// TIA Portal V17 export
// export: Created 2025-03-07T09:24:32.6237895Z, ExportSetting WithDefaults, DisplayName Totally Integrated Automation Portal, DisplayVersion V17 Update 8, DisplayName TIA Portal Openness, DisplayVersion V17 Update 8, DisplayName TIA Portal Version Control Interface, DisplayVersion V17, DisplayName SINAMICS Startdrive Advanced, DisplayVersion V17 SP2, DisplayName SINAMICS Startdrive G110M, G120, G120C, G120D, G120P, G115D, DisplayVersion V17 SP2, DisplayName SINAMICS Startdrive G130, G150, S120, S150, SINAMICS MV, S210, DisplayVersion V17 SP2, DisplayName STEP 7 Professional, DisplayVersion V17 Update 8, DisplayName SINUMERIK ONE STEP 7 Toolbox, DisplayVersion V17 Update 12, DisplayName SINUMERIK 840D sl STEP 7 Toolbox, DisplayVersion V17 Update 12, DisplayName STEP 7 Safety, DisplayVersion V17 Update 6, DisplayName WinCC Advanced, DisplayVersion V17 Update 8
VAR_GLOBAL   // PLC tag table "TAGS_IO_STIRRERS_CLADDING"
   "//////////_STIRRER_UNIT_01_HOPPER_1_//////////" AT %M500.0 : Bool;
   "//////////_STIRRER_UNIT_01_HOPPER_2_//////////" AT %M600.0 : Bool;
   "//////////_STIRRER_UNIT_02_HOPPER_1_//////////" AT %M2000.0 : Bool;
   "//////////_STIRRER_UNIT_02_HOPPER_2_//////////" AT %M800.0 : Bool;
   "//////////_STIRRER_UNIT_02_HOPPER_3_//////////" AT %M900.0 : Bool;
   U01_HPPR_1_STRR_ACTUAL_PHASE_CURRENT_FILTERED_INPUT AT %ID3016 : DInt;   // UNIT 01 HOPPER 1 STIRRER ACTUAL PHASE CURRENT FILTERED INPUT
   U01_HPPR_1_STRR_ACTUAL_PHASE_CURRENT_INPUT AT %ID3012 : DInt;   // UNIT 01 HOPPER 1 STIRRER ACTUAL PHASE CURRENT INPUT
   U01_HPPR_1_STRR_ACTUAL_POSITION_INPUT AT %ID3008 : DInt;   // UNIT 01 HOPPER 1 STIRRER STIRRER ACTUAL POSITON INPUT
   U01_HPPR_1_STRR_ACTUAL_TEMP_COM AT %IW3023 : Int;   // UNIT 01 HOPPER 1 STIRRER ACTUAL COM CARD TEMPERATURE
   U01_HPPR_1_STRR_ACTUAL_TEMP_POWER AT %IW3021 : Int;   // UNIT 01 HOPPER 1 STIRRER ACTUAL POWER STAGE TEMPERATURE
   U01_HPPR_1_STRR_ACTUAL_VELOCITY_INPUT AT %ID3004 : DInt;   // UNIT 01 HOPPER 1 STIRRER ACTUAL VELOCITY INPUT
   U01_HPPR_1_STRR_ENABLE_POWER_STAGE_OUTPUT AT %QB3005 : Byte;   // UNIT 01 HOPPER 1 STIRRER ENABLE POWER STAGE
   U01_HPPR_1_STRR_ERROR_CODE AT %IW3025 : Int;   // UNIT 01 HOPPER 1 STIRRER ERROR CODE
   U01_HPPR_1_STRR_IO_DIGITAL_OUTPUTS AT %QB3000 : Byte;   // UNIT 01 HOPPER 1 STIRRER IO DIGITAL OUTPUTS
   U01_HPPR_1_STRR_MODE_OF_OPERATION_OUTPUT AT %QB3006 : Byte;   // UNIT 01 HOPPER 1 STIRRER MODE OF OPERATION OUTPUT
   U01_HPPR_1_STRR_MOTOR_ENABLE_1_Q AT %M500.1 : Bool;   // UNIT 01 HOPPER 1 STIRRER MOTOR ENABLE 1 OUTPUT
   U01_HPPR_1_STRR_MOTOR_ENABLE_2_Q AT %M500.2 : Bool;   // UNIT 01 HOPPER 1 STIRRER MOTOR ENABLE 2 OUTPUT
   U01_HPPR_1_STRR_MOTOR_OUT_1 AT %Q3000.1 : Bool;   // UNIT 01 HOPPER 1 STIRRER MOTOR OUT 1
   U01_HPPR_1_STRR_MOTOR_OUT_2 AT %Q3000.2 : Bool;   // UNIT 01 HOPPER 1 STIRRER MOTOR OUT 2
   U01_HPPR_1_STRR_MOTOR_OUT_3 AT %Q3000.3 : Bool;   // UNIT 01 HOPPER 1 STIRRER MOTOR OUT 3
   U01_HPPR_1_STRR_MOTOR_STATUS_ENABLE AT %I3020.0 : Bool;   // UNIT 01 HOPPER 1 STIRRER MOTOR STATUS ENABLED
   U01_HPPR_1_STRR_MOTOR_STATUS_ENABLE_INPUT AT %I3000.0 : Bool;   // UNIT 01 HOPPER 1 STIRRER MOTOR STATUS ENABLE INPUT
   U01_HPPR_1_STRR_MOTOR_STATUS_ERROR AT %I3020.1 : Bool;   // UNIT 01 HOPPER 1 STIRRER MOTOR STATUS ERROR
   U01_HPPR_1_STRR_MOTOR_STATUS_ERROR_INPUT AT %I3000.1 : Bool;   // UNIT 01 HOPPER 1 STIRRER MOTOR STATUS ERROR INPUT
   U01_HPPR_1_STRR_MOTOR_STATUS_REACHED AT %I3020.4 : Bool;   // UNIT 01 HOPPER 1 STIRRER MOTOR STATUS REACHED
   U01_HPPR_1_STRR_MOTOR_STATUS_REACHED_INPUT AT %I3000.4 : Bool;   // UNIT 01 HOPPER 1 STIRRER MOTOR STATUS REACHED INPUT
   U01_HPPR_1_STRR_POWER_STAGE_HW_ENABLE_INPUTS AT %IB3020 : Byte;   // UNIT 01 HOPPER 1 STIRRER POWER STAGE STAGE HW ENABLE INPUTS
   U01_HPPR_1_STRR_STATUS_REGISTER_INPUTS AT %ID3000 : DInt;   // UNIT 01 HOPPER 1 STIRRER STATUS REGISTER INPUTS
   U01_HPPR_2_STRR_ACTUAL_PHASE_CURRENT_FILTERED_INPUT AT %ID3116 : DInt;   // UNIT 01 HOPPER 2 STIRRER ACTUAL PHASE CURRENT FILTERED INPUT
   U01_HPPR_2_STRR_ACTUAL_PHASE_CURRENT_INPUT AT %ID3112 : DInt;   // UNIT 01 HOPPER 2 STIRRER ACTUAL PHASE CURRENT INPUT
   U01_HPPR_2_STRR_ACTUAL_POSITION_INPUT AT %ID3108 : DInt;   // UNIT 01 HOPPER 2 STIRRER STIRRER ACTUAL POSITON INPUT
   U01_HPPR_2_STRR_ACTUAL_TEMP_COM AT %IW3123 : Int;   // UNIT 01 HOPPER 2 STIRRER ACTUAL COM CARD TEMPERATURE
   U01_HPPR_2_STRR_ACTUAL_TEMP_POWER AT %IW3121 : Int;   // UNIT 01 HOPPER 2 STIRRER ACTUAL POWER STAGE TEMPERATURE
   U01_HPPR_2_STRR_ACTUAL_VELOCITY_INPUT AT %ID3104 : DInt;   // UNIT 01 HOPPER 2 STIRRER ACTUAL VELOCITY INPUT
   U01_HPPR_2_STRR_ENABLE_POWER_STAGE_OUTPUT AT %QB3105 : Byte;   // UNIT 01 HOPPER 2 STIRRER ENABLE POWER STAGE
   U01_HPPR_2_STRR_ERROR_CODE AT %IW3125 : Int;   // UNIT 01 HOPPER 2 STIRRER ERROR CODE
   U01_HPPR_2_STRR_IO_DIGITAL_OUTPUTS AT %QB3100 : Byte;   // UNIT 01 HOPPER 2 STIRRER IO DIGITAL OUTPUTS
   U01_HPPR_2_STRR_MODE_OF_OPERATION_OUTPUT AT %QB3106 : Byte;   // UNIT 01 HOPPER 2 STIRRER MODE OF OPERATION OUTPUT
   U01_HPPR_2_STRR_MOTOR_ENABLE_1_Q AT %M600.1 : Bool;   // UNIT 01 HOPPER 2 STIRRER MOTOR ENABLE 1 OUTPUT
   U01_HPPR_2_STRR_MOTOR_ENABLE_2_Q AT %M600.2 : Bool;   // UNIT 01 HOPPER 2 STIRRER MOTOR ENABLE 2 OUTPUT
   U01_HPPR_2_STRR_MOTOR_OUT_1 AT %Q3100.1 : Bool;   // UNIT 01 HOPPER 2 STIRRER MOTOR OUT 1
   U01_HPPR_2_STRR_MOTOR_OUT_2 AT %Q3100.2 : Bool;   // UNIT 01 HOPPER 2 STIRRER MOTOR OUT 2
   U01_HPPR_2_STRR_MOTOR_OUT_3 AT %Q3100.3 : Bool;   // UNIT 01 HOPPER 2 STIRRER MOTOR OUT 3
   U01_HPPR_2_STRR_MOTOR_STATUS_ENABLE AT %I3120.0 : Bool;   // UNIT 01 HOPPER 2 STIRRER MOTOR STATUS ENABLED
   U01_HPPR_2_STRR_MOTOR_STATUS_ENABLE_INPUT AT %I3100.0 : Bool;   // UNIT 01 HOPPER 2 STIRRER MOTOR STATUS ENABLE INPUT
   U01_HPPR_2_STRR_MOTOR_STATUS_ERROR AT %I3120.1 : Bool;   // UNIT 01 HOPPER 2 STIRRER MOTOR STATUS ERROR
   U01_HPPR_2_STRR_MOTOR_STATUS_ERROR_INPUT AT %I3100.1 : Bool;   // UNIT 01 HOPPER 2 STIRRER MOTOR STATUS ERROR INPUT
   U01_HPPR_2_STRR_MOTOR_STATUS_REACHED AT %I3120.4 : Bool;   // UNIT 01 HOPPER 2 STIRRER MOTOR STATUS REACHED
   U01_HPPR_2_STRR_MOTOR_STATUS_REACHED_INPUT AT %I3100.4 : Bool;   // UNIT 01 HOPPER 2 STIRRER MOTOR STATUS REACHED INPUT
   U01_HPPR_2_STRR_POWER_STAGE_HW_ENABLE_INPUTS AT %IB3120 : Byte;   // UNIT 01 HOPPER 2 STIRRER POWER STAGE STAGE HW ENABLE INPUTS
   U01_HPPR_2_STRR_STATUS_REGISTER_INPUTS AT %ID3100 : DInt;   // UNIT 01 HOPPER 2 STIRRER STATUS REGISTER INPUTS
   U01_HPPR_2_STRR_VEL_TARGET_VALUE_OUTPUT AT %QD3101 : DInt;   // UNIT 01 HOPPER 2 STIRRER VELOCITY TARGET VALUE OUTPUT
   U01_HPPR1_STRR_VEL_TARGET_VALUE_OUTPUT AT %QD3001 : DInt;   // UNIT 01 HOPPER 1 STIRRER VELOCITY TARGET VALUE OUTPUT
   U02_HPPR_1_STRR_ACTUAL_PHASE_CURRENT_FILTERED_INPUT AT %ID3216 : DInt;   // UNIT 02 HOPPER 1 STIRRER ACTUAL PHASE CURRENT FILTERED INPUT
   U02_HPPR_1_STRR_ACTUAL_PHASE_CURRENT_INPUT AT %ID3212 : DInt;   // UNIT 02 HOPPER 1 STIRRER ACTUAL PHASE CURRENT INPUT
   U02_HPPR_1_STRR_ACTUAL_POSITION_INPUT AT %ID3208 : DInt;   // UNIT 02 HOPPER 1 STIRRER STIRRER ACTUAL POSITON INPUT
   U02_HPPR_1_STRR_ACTUAL_TEMP_COM AT %IW3223 : Int;   // UNIT 02 HOPPER 1 STIRRER ACTUAL COM CARD TEMPERATURE
   U02_HPPR_1_STRR_ACTUAL_TEMP_POWER AT %IW3221 : Int;   // UNIT 02 HOPPER 1 STIRRER ACTUAL POWER STAGE TEMPERATURE
   U02_HPPR_1_STRR_ACTUAL_VELOCITY_INPUT AT %ID3204 : DInt;   // UNIT 02 HOPPER 1 STIRRER ACTUAL VELOCITY INPUT
   U02_HPPR_1_STRR_ENABLE_POWER_STAGE_OUTPUT AT %QB3205 : Byte;   // UNIT 02 HOPPER 1 STIRRER ENABLE POWER STAGE
   U02_HPPR_1_STRR_ERROR_CODE AT %IW3225 : Int;   // UNIT 02 HOPPER 1 STIRRER ERROR CODE
   U02_HPPR_1_STRR_IO_DIGITAL_OUTPUTS AT %QB3200 : Byte;   // UNIT 02 HOPPER 1 STIRRER IO DIGITAL OUTPUTS
   U02_HPPR_1_STRR_MODE_OF_OPERATION_OUTPUT AT %QB3206 : Byte;   // UNIT 02 HOPPER 1 STIRRER MODE OF OPERATION OUTPUT
   U02_HPPR_1_STRR_MOTOR_ENABLE_1_Q AT %M700.1 : Bool;   // UNIT 02 HOPPER 1 STIRRER MOTOR ENABLE 1 OUTPUT
   U02_HPPR_1_STRR_MOTOR_ENABLE_2_Q AT %M700.2 : Bool;   // UNIT 02 HOPPER 1 STIRRER MOTOR ENABLE 2 OUTPUT
   U02_HPPR_1_STRR_MOTOR_OUT_1 AT %Q3200.1 : Bool;   // UNIT 02 HOPPER 1 STIRRER MOTOR OUT 1
   U02_HPPR_1_STRR_MOTOR_OUT_2 AT %Q3200.2 : Bool;   // UNIT 02 HOPPER 1 STIRRER MOTOR OUT 2
   U02_HPPR_1_STRR_MOTOR_OUT_3 AT %Q3200.3 : Bool;   // UNIT 02 HOPPER 1 STIRRER MOTOR OUT 3
   U02_HPPR_1_STRR_MOTOR_STATUS_ENABLE AT %I3220.0 : Bool;   // UNIT 02 HOPPER 1 STIRRER MOTOR STATUS ENABLED
   U02_HPPR_1_STRR_MOTOR_STATUS_ENABLE_INPUT AT %I3200.0 : Bool;   // UNIT 02 HOPPER 1 STIRRER MOTOR STATUS ENABLE INPUT
   U02_HPPR_1_STRR_MOTOR_STATUS_ERROR AT %I3220.1 : Bool;   // UNIT 02 HOPPER 1 STIRRER MOTOR STATUS ERROR
   U02_HPPR_1_STRR_MOTOR_STATUS_ERROR_INPUT AT %I3200.1 : Bool;   // UNIT 02 HOPPER 1 STIRRER MOTOR STATUS ERROR INPUT
   U02_HPPR_1_STRR_MOTOR_STATUS_REACHED AT %I3220.4 : Bool;   // UNIT 02 HOPPER 1 STIRRER MOTOR STATUS REACHED
   U02_HPPR_1_STRR_MOTOR_STATUS_REACHED_INPUT AT %I3200.4 : Bool;   // UNIT 02 HOPPER 1 STIRRER MOTOR STATUS REACHED INPUT
   U02_HPPR_1_STRR_POWER_STAGE_HW_ENABLE_INPUTS AT %IB3220 : Byte;   // UNIT 02 HOPPER 1 STIRRER POWER STAGE STAGE HW ENABLE INPUTS
   U02_HPPR_1_STRR_STATUS_REGISTER_INPUTS AT %ID3200 : DInt;   // UNIT 02 HOPPER 1 STIRRER STATUS REGISTER INPUTS
   U02_HPPR_1_STRR_VEL_TARGET_VALUE_OUTPUT AT %QD3201 : DInt;   // UNIT 02 HOPPER 1 STIRRER VELOCITY TARGET VALUE OUTPUT
   U02_HPPR_2_STRR_ACTUAL_PHASE_CURRENT_FILTERED_INPUT AT %ID3316 : DInt;   // UNIT 02 HOPPER 2 STIRRER ACTUAL PHASE CURRENT FILTERED INPUT
   U02_HPPR_2_STRR_ACTUAL_PHASE_CURRENT_INPUT AT %ID3312 : DInt;   // UNIT 02 HOPPER 2 STIRRER ACTUAL PHASE CURRENT INPUT
   U02_HPPR_2_STRR_ACTUAL_POSITION_INPUT AT %ID3308 : DInt;   // UNIT 02 HOPPER 2 STIRRER STIRRER ACTUAL POSITON INPUT
   U02_HPPR_2_STRR_ACTUAL_TEMP_COM AT %IW3323 : Int;   // UNIT 02 HOPPER 2 STIRRER ACTUAL COM CARD TEMPERATURE
   U02_HPPR_2_STRR_ACTUAL_TEMP_POWER AT %IW3321 : Int;   // UNIT 02 HOPPER 2 STIRRER ACTUAL POWER STAGE TEMPERATURE
   U02_HPPR_2_STRR_ACTUAL_VELOCITY_INPUT AT %ID3304 : DInt;   // UNIT 02 HOPPER 2 STIRRER ACTUAL VELOCITY INPUT
   U02_HPPR_2_STRR_ENABLE_POWER_STAGE_OUTPUT AT %QB3305 : Byte;   // UNIT 02 HOPPER 2 STIRRER ENABLE POWER STAGE
   U02_HPPR_2_STRR_ERROR_CODE AT %IW3325 : Int;   // UNIT 02 HOPPER 2 STIRRER ERROR CODE
   U02_HPPR_2_STRR_IO_DIGITAL_OUTPUTS AT %QB3300 : Byte;   // UNIT 02 HOPPER 2 STIRRER IO DIGITAL OUTPUTS
   U02_HPPR_2_STRR_MODE_OF_OPERATION_OUTPUT AT %QB3306 : Byte;   // UNIT 02 HOPPER 2 STIRRER MODE OF OPERATION OUTPUT
   U02_HPPR_2_STRR_MOTOR_ENABLE_1_Q AT %M800.1 : Bool;   // UNIT 02 HOPPER 2 STIRRER MOTOR ENABLE 1 OUTPUT
   U02_HPPR_2_STRR_MOTOR_ENABLE_2_Q AT %M800.2 : Bool;   // UNIT 02 HOPPER 2 STIRRER MOTOR ENABLE 2 OUTPUT
   U02_HPPR_2_STRR_MOTOR_OUT_1 AT %Q3300.1 : Bool;   // UNIT 02 HOPPER 2 STIRRER MOTOR OUT 1
   U02_HPPR_2_STRR_MOTOR_OUT_2 AT %Q3300.2 : Bool;   // UNIT 02 HOPPER 2 STIRRER MOTOR OUT 2
   U02_HPPR_2_STRR_MOTOR_OUT_3 AT %Q3300.3 : Bool;   // UNIT 02 HOPPER 2 STIRRER MOTOR OUT 3
   U02_HPPR_2_STRR_MOTOR_STATUS_ENABLE AT %I3320.0 : Bool;   // UNIT 02 HOPPER 2 STIRRER MOTOR STATUS ENABLED
   U02_HPPR_2_STRR_MOTOR_STATUS_ENABLE_INPUT AT %I3300.0 : Bool;   // UNIT 02 HOPPER 2 STIRRER MOTOR STATUS ENABLE INPUT
   U02_HPPR_2_STRR_MOTOR_STATUS_ERROR AT %I3320.1 : Bool;   // UNIT 02 HOPPER 2 STIRRER MOTOR STATUS ERROR
   U02_HPPR_2_STRR_MOTOR_STATUS_ERROR_INPUT AT %I3300.1 : Bool;   // UNIT 02 HOPPER 2 STIRRER MOTOR STATUS ERROR INPUT
   U02_HPPR_2_STRR_MOTOR_STATUS_REACHED AT %I3320.4 : Bool;   // UNIT 02 HOPPER 2 STIRRER MOTOR STATUS REACHED
   U02_HPPR_2_STRR_MOTOR_STATUS_REACHED_INPUT AT %I3300.4 : Bool;   // UNIT 02 HOPPER 2 STIRRER MOTOR STATUS REACHED INPUT
   U02_HPPR_2_STRR_POWER_STAGE_HW_ENABLE_INPUTS AT %IB3320 : Byte;   // UNIT 02 HOPPER 2 STIRRER POWER STAGE STAGE HW ENABLE INPUTS
   U02_HPPR_2_STRR_STATUS_REGISTER_INPUTS AT %ID3300 : DInt;   // UNIT 02 HOPPER 2 STIRRER STATUS REGISTER INPUTS
   U02_HPPR_2_STRR_VEL_TARGET_VALUE_OUTPUT AT %QD3301 : DInt;   // UNIT 02 HOPPER 2 STIRRER VELOCITY TARGET VALUE OUTPUT
   U02_HPPR_3_STRR_ACTUAL_PHASE_CURRENT_FILTERED_INPUT AT %ID3416 : DInt;   // UNIT 02 HOPPER 3 STIRRER ACTUAL PHASE CURRENT FILTERED INPUT
   U02_HPPR_3_STRR_ACTUAL_PHASE_CURRENT_INPUT AT %ID3412 : DInt;   // UNIT 02 HOPPER 3 STIRRER ACTUAL PHASE CURRENT INPUT
   U02_HPPR_3_STRR_ACTUAL_POSITION_INPUT AT %ID3408 : DInt;   // UNIT 02 HOPPER 3 STIRRER STIRRER ACTUAL POSITON INPUT
   U02_HPPR_3_STRR_ACTUAL_TEMP_COM AT %IW3423 : Int;   // UNIT 02 HOPPER 3 STIRRER ACTUAL COM CARD TEMPERATURE
   U02_HPPR_3_STRR_ACTUAL_TEMP_POWER AT %IW3421 : Int;   // UNIT 02 HOPPER 3 STIRRER ACTUAL POWER STAGE TEMPERATURE
   U02_HPPR_3_STRR_ACTUAL_VELOCITY_INPUT AT %ID3404 : DInt;   // UNIT 02 HOPPER 3 STIRRER ACTUAL VELOCITY INPUT
   U02_HPPR_3_STRR_ENABLE_POWER_STAGE_OUTPUT AT %QB3405 : Byte;   // UNIT 02 HOPPER 3 STIRRER ENABLE POWER STAGE
   U02_HPPR_3_STRR_ERROR_CODE AT %IW3425 : Int;   // UNIT 02 HOPPER 3 STIRRER ERROR CODE
   U02_HPPR_3_STRR_IO_DIGITAL_OUTPUTS AT %QB3400 : Byte;   // UNIT 02 HOPPER 3 STIRRER IO DIGITAL OUTPUTS
   U02_HPPR_3_STRR_MODE_OF_OPERATION_OUTPUT AT %QB3406 : Byte;   // UNIT 02 HOPPER 3 STIRRER MODE OF OPERATION OUTPUT
   U02_HPPR_3_STRR_MOTOR_ENABLE_1_Q AT %M900.1 : Bool;   // UNIT 02 HOPPER 3 STIRRER MOTOR ENABLE 1 OUTPUT
   U02_HPPR_3_STRR_MOTOR_ENABLE_2_Q AT %M900.2 : Bool;   // UNIT 02 HOPPER 3 STIRRER MOTOR ENABLE 2 OUTPUT
   U02_HPPR_3_STRR_MOTOR_OUT_1 AT %Q3400.1 : Bool;   // UNIT 02 HOPPER 3 STIRRER MOTOR OUT 1
   U02_HPPR_3_STRR_MOTOR_OUT_2 AT %Q3400.2 : Bool;   // UNIT 02 HOPPER 3 STIRRER MOTOR OUT 2
   U02_HPPR_3_STRR_MOTOR_OUT_3 AT %Q3400.3 : Bool;   // UNIT 02 HOPPER 3 STIRRER MOTOR OUT 3
   U02_HPPR_3_STRR_MOTOR_STATUS_ENABLE AT %I3420.0 : Bool;   // UNIT 02 HOPPER 3 STIRRER MOTOR STATUS ENABLED
   U02_HPPR_3_STRR_MOTOR_STATUS_ENABLE_INPUT AT %I3400.0 : Bool;   // UNIT 02 HOPPER 3 STIRRER MOTOR STATUS ENABLE INPUT
   U02_HPPR_3_STRR_MOTOR_STATUS_ERROR AT %I3420.1 : Bool;   // UNIT 02 HOPPER 3 STIRRER MOTOR STATUS ERROR
   U02_HPPR_3_STRR_MOTOR_STATUS_ERROR_INPUT AT %I3400.1 : Bool;   // UNIT 02 HOPPER 3 STIRRER MOTOR STATUS ERROR INPUT
   U02_HPPR_3_STRR_MOTOR_STATUS_REACHED AT %I3420.4 : Bool;   // UNIT 02 HOPPER 3 STIRRER MOTOR STATUS REACHED
   U02_HPPR_3_STRR_MOTOR_STATUS_REACHED_INPUT AT %I3400.4 : Bool;   // UNIT 02 HOPPER 3 STIRRER MOTOR STATUS REACHED INPUT
   U02_HPPR_3_STRR_POWER_STAGE_HW_ENABLE_INPUTS AT %IB3420 : Byte;   // UNIT 02 HOPPER 3 STIRRER POWER STAGE STAGE HW ENABLE INPUTS
   U02_HPPR_3_STRR_STATUS_REGISTER_INPUTS AT %ID3400 : DInt;   // UNIT 02 HOPPER 3 STIRRER STATUS REGISTER INPUTS
   U02_HPPR_3_STRR_VEL_TARGET_VALUE_OUTPUT AT %QD3401 : DInt;   // UNIT 02 HOPPER 3 STIRRER VELOCITY TARGET VALUE OUTPUT
END_VAR
